// TIA Portal V17 export
// export: Created 2024-09-02T12:50:30.9283526Z, ExportSetting WithDefaults, DisplayName Totally Integrated Automation Portal, DisplayVersion V17, DisplayName TIA Portal Openness, DisplayVersion V17, DisplayName TIA Portal Version Control Interface, DisplayVersion V17, DisplayName STEP 7 Professional, DisplayVersion V17, DisplayName STEP 7 Safety, DisplayVersion V17, DisplayName WinCC Professional, DisplayVersion V17
TYPE "type_OpenCom"
// stored: IsFailsafeCompliant false
   STRUCT
      IN { ExternalWritable := 'False'} : Struct
         Frg { ExternalWritable := 'False'} : Bool;
         Adhoc { ExternalWritable := 'False'} : Bool;
         ID { ExternalWritable := 'False'} : Word;
         Len { ExternalWritable := 'False'} : UDInt;
      END_STRUCT;
      OUT { ExternalWritable := 'False'} : Struct
         Done { ExternalWritable := 'False'} : Bool;
         Busy { ExternalWritable := 'False'} : Bool;
         Error { ExternalWritable := 'False'} : Bool;
         Status { ExternalWritable := 'False'} : Word;
         Len { ExternalWritable := 'False'} : UInt;
      END_STRUCT;
      IO { ExternalWritable := 'False'} : Bool;
      NIO { ExternalWritable := 'False'} : Bool;
      Run { ExternalWritable := 'False'} : Bool;
      ErrStatus { ExternalWritable := 'False'} : Word;
      Len { ExternalWritable := 'False'} : UInt;
      Command { S7_SetPoint := 'True'} : Int := 3;
   END_STRUCT;
END_TYPE
